FUNCTION_BLOCK SS3_ps_Lid_feeder (* Composite FB wrapping other FBs *)
  (* Standard: 61499-2 *)
  (* Version 1.0, 2025-08-24, PS_Transformer_for_Unknown *)
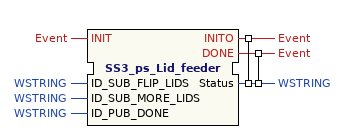
  EVENT_INPUT
    INIT; (* Initialization Request *)
  END_EVENT
  EVENT_OUTPUT
    INITO WITH Status; (* Initialization Confirm *)
    DONE WITH Status; (* Execution Confirmation *)
  END_EVENT
  VAR_INPUT
    ID_SUB_FLIP_LIDS : WSTRING;
    ID_SUB_MORE_LIDS : WSTRING;
    ID_PUB_DONE : WSTRING;
  END_VAR
  VAR_OUTPUT
    Status : WSTRING; (* Output event qualifier *)
  END_VAR
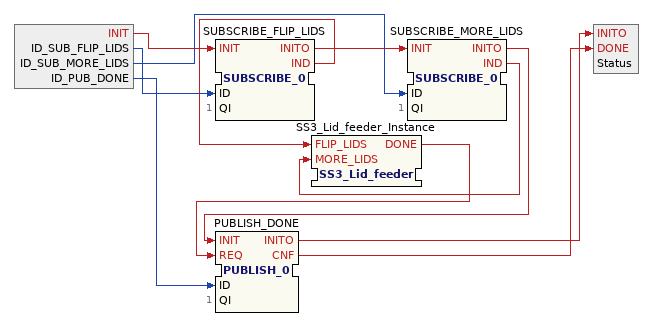
  FBS
    SS3_Lid_feeder_Instance : SS3_Lid_feeder;
    SUBSCRIBE_FLIP_LIDS : SUBSCRIBE_0(QI := 1);
    SUBSCRIBE_MORE_LIDS : SUBSCRIBE_0(QI := 1);
    PUBLISH_DONE : PUBLISH_0(QI := 1);
  END_FBS
  EVENT_CONNECTIONS
    INIT TO SUBSCRIBE_FLIP_LIDS.INIT;
    SUBSCRIBE_FLIP_LIDS.INITO TO SUBSCRIBE_MORE_LIDS.INIT;
    SUBSCRIBE_MORE_LIDS.INITO TO PUBLISH_DONE.INIT;
    PUBLISH_DONE.INITO TO INITO;
    SUBSCRIBE_FLIP_LIDS.IND TO SS3_Lid_feeder_Instance.FLIP_LIDS;
    SUBSCRIBE_MORE_LIDS.IND TO SS3_Lid_feeder_Instance.MORE_LIDS;
    SS3_Lid_feeder_Instance.DONE TO PUBLISH_DONE.REQ;
    PUBLISH_DONE.CNF TO DONE;
  END_CONNECTIONS
  DATA_CONNECTIONS
    ID_SUB_FLIP_LIDS TO SUBSCRIBE_FLIP_LIDS.ID;
    ID_SUB_MORE_LIDS TO SUBSCRIBE_MORE_LIDS.ID;
    ID_PUB_DONE TO PUBLISH_DONE.ID;
  END_CONNECTIONS
END_FUNCTION_BLOCK
